FUNCTION ValidateGeneric : Result
VAR_INPUT
	iToValidate: I_Generic;
END_VAR
VAR
	_err: __SYSTEM.ExceptionCode;
	_iValidate: _I_ValidateGeneric;
END_VAR

IF iToValidate = 0 THEN
	ValidateGeneric := Error;
	RETURN;
END_IF

__TRY
	__QUERYINTERFACE(iToValidate, _iValidate);
	ValidateGeneric := Ok;
__CATCH(_err)
	ValidateGeneric := Error;
__ENDTRY

END_FUNCTION

(* stored: Version 1.1.0.1
   POU ValidateGeneric: Id {70d9f663-5b35-4175-8e0a-2100e2e5c298}, SpecialFunc None *)
